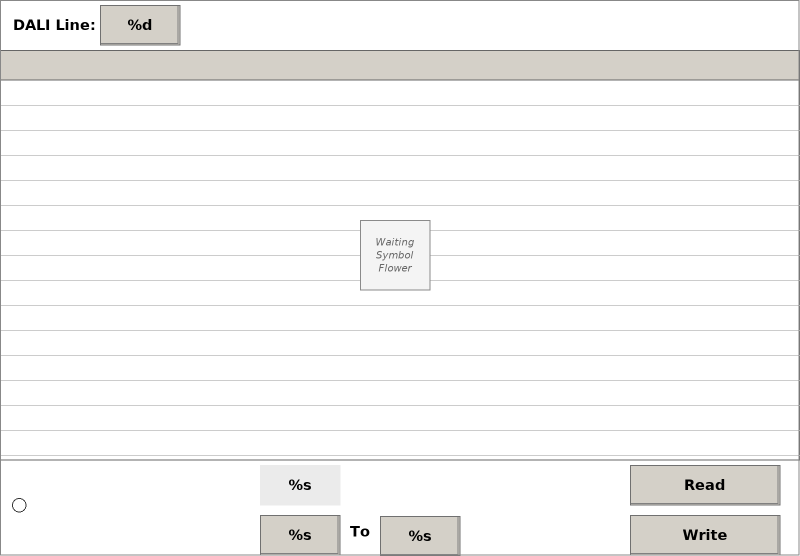
VISUALIZATION Visu_Part102Parameters  // 800x556
    Table (0,50 800x410), data array: DALI_Commissioning.fbPart102Parameters.aParameters
        p1137915858: DALI_Commissioning.fbPart102Parameters.nSelectedAddress
        p3854506369: DALI_Commissioning.fbPart102Parameters.aParameters[INDEX].nShortAddress
        p1892666644: DALI_Commissioning.fbPart102Parameters.aParameters[INDEX].nActualLevel
        p338671338: DALI_Commissioning.fbPart102Parameters.aParameters[INDEX].nMinLevel
        p2170511999: DALI_Commissioning.fbPart102Parameters.aParameters[INDEX].nMaxLevel
        p3723444502: DALI_Commissioning.fbPart102Parameters.aParameters[INDEX].eFadeRate
        p1218418051: DALI_Commissioning.fbPart102Parameters.aParameters[INDEX].eFadeTime
        p746581629: DALI_Commissioning.fbPart102Parameters.aParameters[INDEX].nPowerOnLevel
        p3104783080: DALI_Commissioning.fbPart102Parameters.aParameters[INDEX].nSystemFailureLevel
        p2501879983: DALI_Commissioning.fbPart102Parameters.aParameters[INDEX].nPhysicalMinimum
        p7306298: DALI_Commissioning.fbPart102Parameters.aParameters[INDEX].sDeviceTypes
        Columns.Column.[1].Template: OnMouseClick: write the text variable via Default, min 0, max 254, title "MinLevel"
        Columns.Column.[2].Template: OnMouseClick: write the text variable via Default, min 1, max 254, title "MaxLevel"
        Columns.Column.[3].Template: OnMouseClick: write the text variable via Default, min 0, max 254, title "FadeRate"
        Columns.Column.[4].Template: OnMouseClick: write the text variable via Default, min 1, max 15, title "Fade Rate"
        Columns.Column.[5].Template: OnMouseClick: write the text variable via Default, min 0, max 15, title "Fade Time"
        Columns.Column.[6].Template: OnMouseClick: write the text variable via Default, min 1, max 254, title "Power On Level"
        Columns.Column.[7].Template: OnMouseClick: write the text variable via Default, min 0, max 255, title "System Failure Level"
    RadioButton (10,455 254x100), variable: DALI_Commissioning.fbPart102Parameters.nAddressRange
        Areas[0]: Text=Single Short Address
        Areas[1]: Text=Short Address Range
    Textfield (335,516 50x31), "To"
    Button (630,465 150x40), "Read"
        OnMouseClick: execute { DALI_Commissioning.fbPart102Parameters.bRead := TRUE; }
    Button (630,515 150x40), "Write"
        OnMouseClick: execute { DALI_Commissioning.fbPart102Parameters.bWrite := TRUE; }
    Button (260,515 80x40), "%s", text variable: DALI_Commissioning.fbPart102Parameters.nStartAddress
        OnMouseClick: write the text variable via Default, min 0, max 63, title "Insert Short Address"
    Button (380,516 80x40), "%s", text variable: DALI_Commissioning.fbPart102Parameters.nEndAddress
        OnMouseClick: write the text variable via Default, min 0, max 63, title "Insert Short Address"
    Textfield (260,465 80x40), "%s", tooltip "Please select the desired Short Address in the table above.", text variable: DALI_Commissioning.fbPart102Parameters.nSelectedAddress
    WaitingSymbolFlower (360,220 70x70), invisible if: DALI_Commissioning.fbPart102Parameters.bHideWaitSymbol
    Group (10,5 170x40)
        Textfield (0,0 110x40), "DALI Line:"
        Button (90,0 80x40), "%d", text variable: GVL_Internal.nDALILine
            OnMouseClick: write the text variable via Default, min 1, max 10, title "Choose line"
END_VISUALIZATION

// ---- POUs/DALI/DALI_Setup/VISUs/Visu_DALICommissioning/Visu_Part300GenericDevice.TcVIS
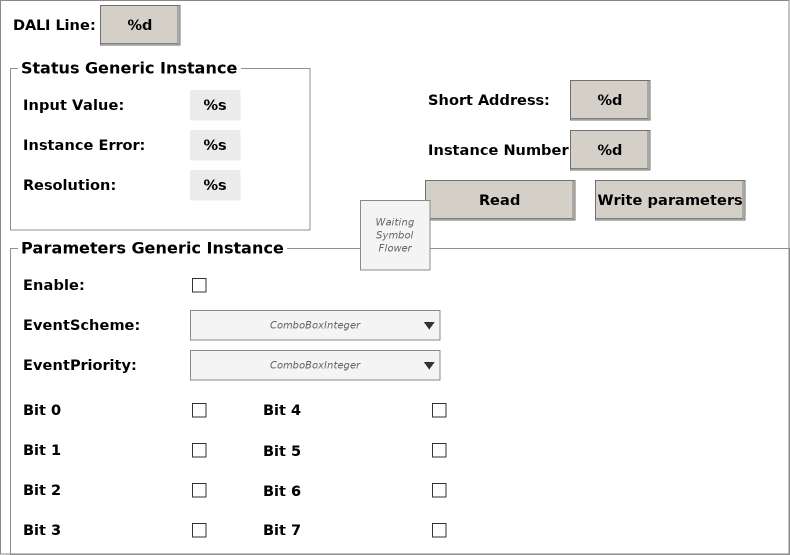
VISUALIZATION Visu_Part300GenericDevice  // 790x555
    GroupBox (10,240 780x315), "Parameters Generic Instance"
        Textfield (10,30 150x30), "Enable:"
        Checkbox (180,30 30x30), variable: DALI_Commissioning.fbPart300GenericDevice.bEnable
        Textfield (10,110 150x30), "EventPriority:"
        Textfield (10,195 100x30), "Bit 1"
        Textfield (10,155 100x30), "Bit 0"
        Checkbox (180,155 30x30), variable: DALI_Commissioning.fbPart300GenericDevice.bBit0
        Checkbox (180,195 30x30), variable: DALI_Commissioning.fbPart300GenericDevice.bBit1
        Textfield (10,235 100x30), "Bit 2"
        Textfield (250,155 100x30), "Bit 4"
        Textfield (250,196 100x30), "Bit 5"
        Checkbox (420,195 30x30), variable: DALI_Commissioning.fbPart300GenericDevice.bBit5
        Checkbox (420,155 30x30), variable: DALI_Commissioning.fbPart300GenericDevice.bBit4
        Checkbox (180,275 30x30), variable: DALI_Commissioning.fbPart300GenericDevice.bBit3
        Checkbox (180,235 30x30), variable: DALI_Commissioning.fbPart300GenericDevice.bBit2
        ComboBoxInteger (180,70 250x30), variable: DALI_Commissioning.fbPart300GenericDevice.eEventScheme, text list: 'EventScheme'
        Textfield (10,70 150x30), "EventScheme:"
        Textfield (250,236 100x30), "Bit 6"
        ComboBoxInteger (180,110 250x30), variable: DALI_Commissioning.fbPart300GenericDevice.eEventPriority, text list: 'EventPriority'
        Textfield (10,275 100x30), "Bit 3"
        Checkbox (420,235 30x30), variable: DALI_Commissioning.fbPart300GenericDevice.bBit6
        Checkbox (420,275 30x30), variable: DALI_Commissioning.fbPart300GenericDevice.bBit7
        Textfield (250,275 100x30), "Bit 7"
    GroupBox (10,60 300x170), "Status Generic Instance"
        Textfield (180,30 50x30), "%s", text variable: DALI_Commissioning.fbPart300GenericDevice.nInputValue
        Textfield (180,70 50x30), "%s", text variable: DALI_Commissioning.fbPart300GenericDevice.nInstanceError
        Textfield (180,110 50x30), "%s", text variable: DALI_Commissioning.fbPart300GenericDevice.nResolution
        Textfield (10,30 160x30), "Input Value:"
        Textfield (10,70 160x30), "Instance Error:"
        Textfield (10,110 160x30), "Resolution:"
    Button (425,180 150x40), "Read"
        OnMouseClick: execute { DALI_Commissioning.fbPart300GenericDevice.bRead := TRUE; }
    WaitingSymbolFlower (360,200 70x70), invisible if: DALI_Commissioning.fbPart300GenericDevice.bHideWaitSymbol
    Button (595,180 150x40), "Write parameters"
        OnMouseClick: execute { DALI_Commissioning.fbPart300GenericDevice.bWrite := TRUE; }
    Textfield (425,130 150x40), "Instance Number:"
    Textfield (425,80 150x40), "Short Address:"
    Button (570,80 80x40), "%d", text variable: DALI_Commissioning.fbPart300GenericDevice.nAddress
        OnMouseClick: write the text variable via Default, min 0, max 63, title "Insert Short Address"
    Button (570,130 80x40), "%d", text variable: DALI_Commissioning.fbPart300GenericDevice.nInstanceAddress
        OnMouseClick: write the text variable via Default, min 0, max 31, title "Insert instance number"
    Group (10,5 170x40)
        Textfield (0,0 110x40), "DALI Line:"
        Button (90,0 80x40), "%d", text variable: GVL_Internal.nDALILine
            OnMouseClick: write the text variable via Default, min 1, max 10, title "Choose line"
END_VISUALIZATION

// ---- POUs/DALI/DALI_Setup/VISUs/Visu_DALICommissioning/Visu_Part304LightSensor.TcVIS
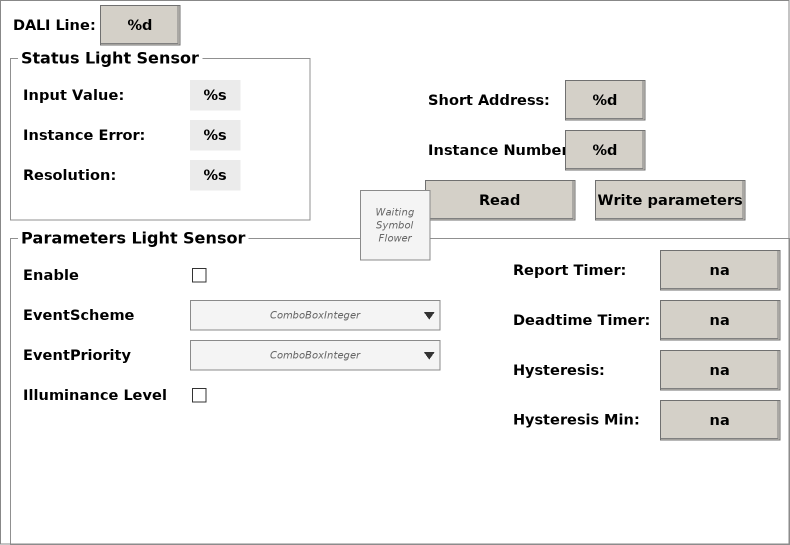
VISUALIZATION Visu_Part304LightSensor  // 790x545
    GroupBox (10,230 780x315), "Parameters Light Sensor"
        Button (650,120 120x40), "%d %%", text variable: DALI_Commissioning.fbPart304LightSensor.nHysteresis
            OnMouseClick: write the text variable via Default, min 0, max 25, title "Insert value for hysteresis"
        Button (650,120 120x40), "na", invisible if: not DALI_Commissioning.fbPart304LightSensor.bNoHysteresis, input disabled if: not DALI_Commissioning.fbPart304LightSensor.bNoHysteresis
        Button (650,170 120x40), "%d", text variable: DALI_Commissioning.fbPart304LightSensor.nHysteresisMin
            OnMouseClick: write the text variable via Default, min 0, max 255, title "Insert value for hysteresis min"
        Button (650,170 120x40), "na", invisible if: not DALI_Commissioning.fbPart304LightSensor.bNoHysteresisMin, input disabled if: not DALI_Commissioning.fbPart304LightSensor.bNoHysteresisMin
        Button (650,20 120x40), "%d s", text variable: DALI_Commissioning.fbPart304LightSensor.nReport
            OnMouseClick: write the text variable via Default, min 0, max 255, title "Insert value for report timer"
        Button (650,70 120x40), "%d ms", text variable: DALI_Commissioning.fbPart304LightSensor.nDeadtime
            OnMouseClick: write the text variable via Default, min 0, max 12750, title "Insert value for deadtime timer"
        Button (650,70 120x40), "na", invisible if: not DALI_Commissioning.fbPart304LightSensor.bNoDeadtimeTimer, input disabled if: not DALI_Commissioning.fbPart304LightSensor.bNoDeadtimeTimer
        Button (650,20 120x40), "na", invisible if: not DALI_Commissioning.fbPart304LightSensor.bNoReportTimer, input disabled if: not DALI_Commissioning.fbPart304LightSensor.bNoReportTimer
        Textfield (500,175 145x29), "Hysteresis Min:"
        Textfield (500,125 145x30), "Hysteresis:"
        Textfield (500,25 145x30), "Report Timer:"
        Textfield (500,75 145x30), "Deadtime Timer:"
        Textfield (10,30 150x30), "Enable"
        Checkbox (180,30 30x30), variable: DALI_Commissioning.fbPart304LightSensor.bEnable
        Textfield (10,70 150x30), "EventScheme"
        Textfield (10,150 150x30), "Illuminance Level"
        ComboBoxInteger (180,70 250x30), variable: DALI_Commissioning.fbPart304LightSensor.eEventScheme, text list: 'EventScheme'
        Checkbox (180,150 30x30), variable: DALI_Commissioning.fbPart304LightSensor.bIlluminanceLevel
        Textfield (10,110 150x30), "EventPriority"
        ComboBoxInteger (180,110 250x30), variable: DALI_Commissioning.fbPart304LightSensor.eEventPriority, text list: 'EventPriority'
    GroupBox (10,50 300x170), "Status Light Sensor"
        Textfield (10,30 160x30), "Input Value:"
        Textfield (10,70 160x30), "Instance Error:"
        Textfield (10,110 160x30), "Resolution:"
        Textfield (180,30 50x30), "%s", text variable: DALI_Commissioning.fbPart304LightSensor.nInputValue
        Textfield (180,70 50x30), "%s", text variable: DALI_Commissioning.fbPart304LightSensor.nInstanceError
        Textfield (180,110 50x30), "%s", text variable: DALI_Commissioning.fbPart304LightSensor.nResolution
    Button (425,180 150x40), "Read"
        OnMouseClick: execute { DALI_Commissioning.fbPart304LightSensor.bRead := TRUE; }
    WaitingSymbolFlower (360,190 70x70), invisible if: DALI_Commissioning.fbPart304LightSensor.bHideWaitSymbol
    Button (595,180 150x40), "Write parameters"
        OnMouseClick: execute { DALI_Commissioning.fbPart304LightSensor.bWrite := TRUE; }
    Textfield (425,80 130x40), "Short Address:"
    Button (565,80 80x40), "%d", text variable: DALI_Commissioning.fbPart304LightSensor.nAddress
        OnMouseClick: write the text variable via Default, min 0, max 63, title "Insert Short Address"
    Textfield (425,130 150x40), "Instance Number:"
    Button (565,130 80x40), "%d", text variable: DALI_Commissioning.fbPart304LightSensor.nInstanceAddress
        OnMouseClick: write the text variable via Default, min 0, max 31, title "Insert instance number"
    Group (10,5 170x40)
        Textfield (0,0 110x40), "DALI Line:"
        Button (90,0 80x40), "%d", text variable: GVL_Internal.nDALILine
            OnMouseClick: write the text variable via Default, min 1, max 10, title "Choose line"
END_VISUALIZATION
